// TIA Portal V16 export
// export: Created 2023-03-29T11:03:38.9872883Z, ExportSetting WithDefaults, DisplayName Totally Integrated Automation Portal, DisplayVersion V16 Update 6, DisplayName TIA Portal Version Control Interface, DisplayVersion V16 Update 2, DisplayName TIA Portal Openness, DisplayVersion V16 Update 6, DisplayName STEP 7 Professional, DisplayVersion V16 Update 6, DisplayName STEP 7 Safety, DisplayVersion V16, DisplayName WinCC Advanced, DisplayVersion V16 Update 6
DATA_BLOCK "alarm_petli-rtu_tcp_DB"   // DB66
AUTHOR : rtecmer
VERSION : 0.1
// stored: AutoNumber true, DBAccessibleFromOPCUA true, InstanceOfName alarm_petli-rtu_tcp, InstanceOfType FB
"alarm_petli-rtu_tcp"
BEGIN
END_DATA_BLOCK
